(******************************************************************************************************************************************)
(****************************				           Reset Function Part                                                 *****************************)
(******************************************************************************************************************************************)
IF xReset THEN
	xReset:=FALSE;
	xSetEnd:=TRUE;
END_IF;
(******************************************************************************************************************************************)
(****************************				              Error Controlling Part                                            *****************************)
(******************************************************************************************************************************************)
IF (xSetError OR T_Station.TControl.xError) AND NOT(xSetEnd) THEN
	IF NOT(xInitError) THEN
		iStepError:=100;
		xInitError:=TRUE;
		IF NOT(xSetError) THEN
			xSetError:=TRUE;
			xSetTmpError:=FALSE;
		ELSE
			xSetTmpError:=TRUE;
		END_IF;
	END_IF;
	CASE iStepError OF
		100:	IF T_Station.TControl.xError THEN
				diErrorNr:=T_Station.TControl.diErrorNr;
			END_IF;
			IF xSetTmpError THEN
				diErrorNr:=diTmpErrNr;
			END_IF;
			iStepError:=200;
		200:	IF xSetTmpError THEN
				xSetTmpError:=FALSE;
				xStopFctStation1:=FALSE;
				iStepError:=300;
			ELSE
				IF NOT(T_Station.TControl.xError) AND NOT(T_Station.TControl.xEnd) THEN
					IF (T_Station.TControl.iFunctNr = 1) THEN
						T_Station.TControl.xStop:=TRUE;
						xStopFctStation1:=TRUE;
					ELSE
						xStopFctStation1:=FALSE;
					END_IF;
				END_IF;
				iStepError:=300;
			END_IF;
		300:	IF xStopFctStation1 THEN
				IF NOT(T_Station.TControl.xStop) THEN
					xStopFctStation1:=FALSE;
				END_IF;
			END_IF;
			IF NOT(xStopFctStation1) THEN
				xError:=TRUE;
				iStepError:=400;
			END_IF;
		400:	IF xQuitErr THEN
				T_Station.TControl.xQuitError:=T_Station.TControl.xError;
				iStepError:=500;
			END_IF;
		500: IF NOT(T_Station.TControl.xQuitError) THEN
				xSetEnd:=TRUE;
			END_IF;
	END_CASE;
END_IF;
(******************************************************************************************************************************************)
(****************************				              Main Controlling Part                                            *****************************)
(******************************************************************************************************************************************)
IF (xStart OR xStartMainCtr) AND NOT(xSetEnd) AND NOT(xSetError) THEN
	IF NOT (xInitMainCtr) THEN
		iStepPrc:=10;
		xInitMainCtr:=TRUE;
		xStartMainCtr:=TRUE;
		xStart:=FALSE;
		xEnd:=FALSE;
		xSetEndPrc:=FALSE;
		iTmpFunctionNr:=1;
		xAbord:=FALSE;
		T_ExchgParam.T_InfoValueCommon.rActualWireFeedPosition:=0.0;
		T_ExchgParam.T_InfoValueCommon.rActualWireFeedSpeed:=0.0;
	END_IF;
	IF xStop AND NOT(xTmpStop) THEN
		xTmpStop:=TRUE;
		iStepStop:=1;
	END_IF;
	IF xTmpStop THEN
		CASE iStepStop OF
		1:	IF NOT(T_Station.TControl.xEnd) THEN
				T_Station.TControl.xStop:=TRUE;
				iStepStop:=10;
			ELSE
				iStepStop:=20;
			END_IF;
		10:	IF NOT(T_Station.TControl.xStop) THEN
				iStepStop:=20;
			END_IF;
		20:	IF NOT(T_Station.TControl.xStart) AND T_Station.TControl.xEnd THEN
				T_Station.TControl.iFunctNr:=4;
				T_Station.TControl.xStart:=TRUE;
				T_Station.THardware.TAxisGrindFeeder.T_CtrleSingle.lrAcceleration:=T_NovRAMData.T_Standard.T_TeachINGrindFeeder.rAcceleration;
				T_Station.THardware.TAxisGrindFeeder.T_CtrleSingle.lrDecceleration:=T_NovRAMData.T_Standard.T_TeachINGrindFeeder.rDeceleration;
				T_Station.THardware.TAxisGrindFeeder.T_CtrleSingle.lrPosition:=	T_NovRAMData.T_ProcessImageData.T_ProcessPara.rToolDiameterProcess +
																			T_NovRAMData.T_ProcessImageData.T_ProcessPara.rSecurityPosGrindFeedProcess;
				T_Station.THardware.TAxisGrindFeeder.T_CtrleSingle.lrVelocity:=T_NovRAMData.T_ProcessImageData.T_ProcessPara.rSpeedBackwardGrindFeed;
				iStepStop:=30;
			END_IF;
		(* Check Active Movement of the Axis *)
		30:	IF NOT(T_Station.TControl.xStart) AND T_Station.TControl.xEnd THEN
				T_Station.TControl.iFunctNr:=18;	(* Check Axis Movement, and stop it if moves *)
				T_Station.TControl.xStart:=TRUE;
				iStepStop:=40;
			END_IF;
		40:	IF NOT(T_Station.TControl.xStart) AND T_Station.TControl.xEnd THEN
				xStartMainPrc:=FALSE;
				xInitStep:=FALSE;
				iStepPrc:=0;
				xSetEnd:=TRUE;
				RETURN;
			END_IF;
		END_CASE;
		RETURN;
	END_IF;
	IF NOT(xStartMainPrc) THEN
		xStartMainPrc:=TRUE;
	END_IF;
END_IF;
(******************************************************************************************************************************************)
(****************************				             Main Procedure Part                                             *****************************)
(******************************************************************************************************************************************)
IF xStartProcess THEN
	TONStartTimer(IN:=TRUE,PT:=T#1s);
	IF TONStartTimer.Q THEN
		TONStartTimer(IN:=FALSE);
		IF (T_ExchgParam.T_InfoValueCommon.tAutoTimeLeft >= T#1s) THEN
			T_ExchgParam.T_InfoValueCommon.tAutoTimeLeft:=T_ExchgParam.T_InfoValueCommon.tAutoTimeLeft - T#1s;
		ELSE
			T_ExchgParam.T_InfoValueCommon.tAutoTimeLeft:=T#0s;
		END_IF;
	END_IF;
	tStepTime:=T_ExchgParam.T_InfoValueCommon.tAutoTimeTotal / 100;
	TONStartTimer1(IN:=TRUE,PT:=tStepTime);
	IF TONStartTimer1.Q THEN
		TONStartTimer1(IN:=FALSE);
		T_ExchgParam.T_InfoValueCommon.bProgressbarToolCalibration:=T_ExchgParam.T_InfoValueCommon.bProgressbarToolCalibration + 1;
		IF (T_ExchgParam.T_InfoValueCommon.bProgressbarToolCalibration >= 100) THEN
			T_ExchgParam.T_InfoValueCommon.bProgressbarToolCalibration:=100;
		END_IF;
	END_IF;
ELSE
	TONStartTimer(IN:=FALSE);
	TONStartTimer1(IN:=FALSE);
END_IF;
IF xStartMainPrc AND NOT(xSetEnd) AND NOT(xSetError) THEN
	CASE iStepPrc OF
		(* Check first if the ToolCalibration is available to start it *)
		10:	T_Station.THardware.TAxisToolLeft.T_CtrleSingle.lrAcceleration:=T_NovRAMData.T_Standard.T_TeachINToolLeft.rAcceleration;
			T_Station.THardware.TAxisToolLeft.T_CtrleSingle.lrDecceleration:=T_NovRAMData.T_Standard.T_TeachINToolLeft.rDeceleration;
			T_Station.THardware.TAxisToolCenter.T_CtrleSingle.lrAcceleration:=T_NovRAMData.T_Standard.T_TeachINToolCenter.rAcceleration;
			T_Station.THardware.TAxisToolCenter.T_CtrleSingle.lrDecceleration:=T_NovRAMData.T_Standard.T_TeachINToolCenter.rDeceleration;
			T_Station.THardware.TAxisToolRight.T_CtrleSingle.lrAcceleration:=T_NovRAMData.T_Standard.T_TeachINToolRight.rAcceleration;
			T_Station.THardware.TAxisToolRight.T_CtrleSingle.lrDecceleration:=T_NovRAMData.T_Standard.T_TeachINToolRight.rDeceleration;
			T_Station.THardware.TAxisToolFeeder.T_CtrleSingle.lrAcceleration:=T_NovRAMData.T_Standard.T_TeachINToolFeeder.rAcceleration;
			T_Station.THardware.TAxisToolFeeder.T_CtrleSingle.lrDecceleration:=T_NovRAMData.T_Standard.T_TeachINToolFeeder.rDeceleration;
			T_Station.THardware.TAxisGrindFeeder.T_CtrleSingle.lrAcceleration:=T_NovRAMData.T_Standard.T_TeachINGrindFeeder.rAcceleration;
			T_Station.THardware.TAxisGrindFeeder.T_CtrleSingle.lrDecceleration:=T_NovRAMData.T_Standard.T_TeachINGrindFeeder.rDeceleration;
			(* Only for MicroRod, check if the tool is clamped *)
			IF xMicroRodActive THEN
				(*22.12.2009: KFS	{ *)
				(*
				IF T_Station.THardware.TCylToolTension.T_CtrleCyl.xStatePosOn THEN
					xSetError:=TRUE;
					diTmpErrNr:=2;			(* Tool is not clamped *)
				END_IF;
				*)
				(*Added control if all cylinder for the tool are activated*)
				IF T_Station.THardware.TCylToolTension.T_CtrleCyl.xStatePosOn OR
				     T_Station.THardware.TCylToolLeftActive.T_CtrleCyl.T_Standard.xActivOn OR
 				     T_Station.THardware.TCylToolRightActive.T_CtrleCyl.T_Standard.xActivOn  OR
				   (* T_Station.THardware.TCylToolCenterActive.T_CtrleCyl.T_Standard.xActivOn OR*)	(* IGS auskommentiert, diesen Zyl gibts auf der M3 nicht *)
				     NOT(T_Station.THardware.TCylToolPrismaLeftActive.T_CtrleCyl.T_Standard.xActivOn) OR
				     NOT(T_Station.THardware.TCylToolPrismaRightActive.T_CtrleCyl.T_Standard.xActivOn) 	THEN
					xSetError:=TRUE;
					diTmpErrNr:=2;			(* Tool is not clamped *)
				END_IF;
				(*22.12.2009: KFS	} *)
			END_IF;
			(* Only for MicroRod, check if the Machine is referenced *)
			IF xMicroRodActive THEN
				IF NOT(T_Station.TControl.xReferenced) THEN
					xSetError:=TRUE;
					diTmpErrNr:=1;	(* Machine is not referenced *)
					RETURN;
				END_IF;
			END_IF;
			xStartMainPrc:=FALSE;
			xInitStep:=FALSE;
			iStepPrc:=11;
		(* Set the ToolTension force *)
		11:	IF NOT(xInitStep) THEN
				xInitStep:=TRUE;
				T_Station.THardware.TCylToolTension.T_CtrleCyl.iFunction:=2;	(* activate the ToolTension *)
				T_Station.THardware.TCylToolTension.T_CtrleCyl.T_AnalogCylinder.rForceIn:=T_NovRAMData.T_ProcessImageData.T_ProcessPara.rToolTensionProcess;
				IF xMicroRodActive THEN
					T_Station.THardware.TCylToolTension.T_Config.tDelayOn:=T#1s;
				ELSE
					T_Station.THardware.TCylToolTension.T_Config.tDelayOn:=T#0s;
				END_IF;
				T_Station.THardware.TCylToolTension.T_CtrleCyl.xExecute:=TRUE;
			END_IF;
			IF NOT(T_Station.THardware.TCylToolTension.T_CtrleCyl.xExecute) AND T_Station.THardware.TCylToolTension.T_CtrleCyl.xDone THEN
				(* Only for MicroRod, check if the tool is clamped *)
				IF xMicroRodActive THEN
					IF T_Station.THardware.TCylToolTension.T_CtrleCyl.xStatePosOn THEN
						xSetError:=TRUE;
						diTmpErrNr:=2;			(* Tool is not clamped *)
						RETURN;
					END_IF;
				END_IF;
				iStepPrc:=20;
				xStartMainPrc:=FALSE;
				xInitStep:=FALSE;
			END_IF;
		(* Switch First all Axis the power supply on *)
		20:	IF NOT(xInitStep) THEN
				xInitStep:=TRUE;
				T_Station.TControl.iFunctNr:=16;
				T_Station.TControl.xStart:=TRUE;
			END_IF;
			IF NOT(T_Station.TControl.xStart) AND T_Station.TControl.xEnd THEN
				iStepPrc:=30;
				xStartMainPrc:=FALSE;
				xInitStep:=FALSE;
				iTmpStationFunctionNr:=6;
				T_Station.THardware.TAxisToolLeft.T_CtrleSingle.rSetPosition:=0.0;
				T_Station.THardware.TAxisToolCenter.T_CtrleSingle.rSetPosition:=0.0;
				T_Station.THardware.TAxisToolRight.T_CtrleSingle.rSetPosition:=0.0;
				T_Station.THardware.TAxisToolFeeder.T_CtrleSingle.rSetPosition:=0.0;
			END_IF;
		(* Reset the Position of the Axis *)
		30:	IF NOT(xInitStep) THEN
				xInitStep:=TRUE;
				(* 6=ToolLeft, 7=ToolCenter, 8=ToolRight, 9=ToolFeeder *)
				T_Station.TControl.iFunctNr:=iTmpStationFunctionNr;
				T_Station.TControl.xStart:=TRUE;
			END_IF;
			IF NOT(T_Station.TControl.xStart) AND T_Station.TControl.xEnd THEN
				iTmpStationFunctionNr:=iTmpStationFunctionNr + 1;
				IF NOT(xMicroRodActive) AND (iTmpStationFunctionNr = 7) THEN
					iTmpStationFunctionNr:=iTmpStationFunctionNr + 1;
				END_IF;
				IF xMicroRodActive AND (iTmpStationFunctionNr = 9) THEN
					iTmpStationFunctionNr:=iTmpStationFunctionNr + 1;
				END_IF;
				xStartMainPrc:=FALSE;
				xInitStep:=FALSE;
				IF (iTmpStationFunctionNr < 10) THEN
					iStepPrc:=30;
				ELSE
					iStepPrc:=40;
				END_IF;
			END_IF;
		(* GrindFeeder Set Absolut to Security Position *)
		40:	IF NOT(xInitStep) THEN
				xInitStep:=TRUE;
				T_Station.TControl.iFunctNr:=4;
				T_Station.TControl.xStart:=TRUE;
				T_Station.THardware.TAxisGrindFeeder.T_CtrleSingle.lrAcceleration:=T_NovRAMData.T_Standard.T_TeachINGrindFeeder.rAcceleration;
				T_Station.THardware.TAxisGrindFeeder.T_CtrleSingle.lrDecceleration:=T_NovRAMData.T_Standard.T_TeachINGrindFeeder.rDeceleration;
				T_Station.THardware.TAxisGrindFeeder.T_CtrleSingle.lrPosition:=	T_NovRAMData.T_ProcessImageData.T_ProcessPara.rToolDiameterProcess +
																			T_NovRAMData.T_ProcessImageData.T_ProcessPara.rSecurityPosGrindFeedProcess;
				T_Station.THardware.TAxisGrindFeeder.T_CtrleSingle.lrVelocity:=T_NovRAMData.T_ProcessImageData.T_ProcessPara.rSpeedBackwardGrindFeed;
			END_IF;
			IF NOT(T_Station.TControl.xStart) AND T_Station.TControl.xEnd THEN
				IF xMicroRodActive THEN
					iStepPrc:=50;
				ELSE
					iStepPrc:=60;
				END_IF;
				xStartMainPrc:=FALSE;
				xInitStep:=FALSE;
			END_IF;
		(* Only for MicroRod-->Set ToolFeed Absolut to the StartPosition and if more cycle than only the first time *)
		50:	IF NOT(xInitStep) THEN
				xInitStep:=TRUE;
				T_Station.TControl.iFunctNr:=14;
				T_Station.TControl.xStart:=TRUE;
				T_Station.THardware.TAxisToolFeeder.T_CtrleSingle.lrAcceleration:=T_NovRAMData.T_Standard.T_TeachINToolFeeder.rAcceleration;
				T_Station.THardware.TAxisToolFeeder.T_CtrleSingle.lrDecceleration:=T_NovRAMData.T_Standard.T_TeachINToolFeeder.rDeceleration;
				T_Station.THardware.TAxisToolFeeder.T_CtrleSingle.lrPosition:=T_NovRAMData.T_ProcessImageData.T_CalibrationPara.rStartPosToolFeedCalib;
				T_Station.THardware.TAxisToolFeeder.T_CtrleSingle.lrVelocity:=T_NovRAMData.T_ProcessImageData.T_ProcessPara.rSpeedStartPosToolFeedProcess;
			END_IF;
			IF NOT(T_Station.TControl.xStart) AND T_Station.TControl.xEnd THEN
				iStepPrc:=60;
				xStartMainPrc:=FALSE;
				xInitStep:=FALSE;
			END_IF;
		(* ToolRotation Start *)
		60:	IF NOT(xInitStep) THEN
				xInitStep:=TRUE;
				T_Station.TControl.iFunctNr:=2;
				T_Station.TControl.xStart:=TRUE;
				(* ToolLeft --> Master *)
				T_Station.THardware.TAxisToolLeft.T_CtrleSingle.lrVelocity:=T_NovRAMData.T_ProcessImageData.T_CalibrationPara.rSpeedToolRotationCalib;
				T_Station.THardware.TAxisToolLeft.T_CtrleSingle.lrAcceleration:=T_NovRAMData.T_Standard.T_TeachINToolLeft.rAcceleration;
				T_Station.THardware.TAxisToolLeft.T_CtrleSingle.lrDecceleration:=T_NovRAMData.T_Standard.T_TeachINToolLeft.rDeceleration;
				IF xMicroRodActive THEN
					(* ToolCenter --> Slave of ToolLeft only by MicroRod *)
					T_Station.THardware.TAxisToolCenter.T_CtrleSingle.lrAcceleration:=T_NovRAMData.T_Standard.T_TeachINToolCenter.rAcceleration;
					T_Station.THardware.TAxisToolCenter.T_CtrleSingle.lrDecceleration:=T_NovRAMData.T_Standard.T_TeachINToolCenter.rDeceleration;
					T_Station.THardware.TAxisToolCenter.T_CtrleSingle.lrGearDivider:=INT_TO_LREAL(T_Station.T_WorkTool.iBaseGearDivider);
					T_Station.THardware.TAxisToolCenter.T_CtrleSingle.lrGearFactor:=(	INT_TO_LREAL(T_Station.T_WorkTool.iBaseGearDivider) /
																					(T_Station.THardware.TAxisToolLeft.T_CtrleSingle.lrGearRatio /
																					T_Station.THardware.TAxisToolCenter.T_CtrleSingle.lrGearRatio)) * -1.0;

					(* ToolRight --> Slave of ToolLeft by MicroWire or Slave of ToolRight by MicroRod *)
					T_Station.THardware.TAxisToolRight.T_CtrleSingle.lrAcceleration:=T_NovRAMData.T_Standard.T_TeachINToolRight.rAcceleration;
					T_Station.THardware.TAxisToolRight.T_CtrleSingle.lrDecceleration:=T_NovRAMData.T_Standard.T_TeachINToolRight.rDeceleration;
					T_Station.THardware.TAxisToolRight.T_CtrleSingle.lrGearDivider:=INT_TO_LREAL(T_Station.T_WorkTool.iBaseGearDivider);
					T_Station.THardware.TAxisToolRight.T_CtrleSingle.lrGearFactor:=	INT_TO_LREAL(T_Station.T_WorkTool.iBaseGearDivider) /
																					(T_Station.THardware.TAxisToolLeft.T_CtrleSingle.lrGearRatio /
																					T_Station.THardware.TAxisToolRight.T_CtrleSingle.lrGearRatio);
				END_IF;

				IF NOT(xMicroRodActive) THEN
					(* ToolRight --> Slave of ToolRight by MicroWire *)
					T_Station.THardware.TAxisToolFeeder.T_CtrleSingle.lrAcceleration:=T_NovRAMData.T_Standard.T_TeachINToolFeeder.rAcceleration;
					T_Station.THardware.TAxisToolFeeder.T_CtrleSingle.lrDecceleration:=T_NovRAMData.T_Standard.T_TeachINToolFeeder.rDeceleration;
					T_Station.THardware.TAxisToolFeeder.T_CtrleSingle.lrGearDivider:=INT_TO_LREAL(T_Station.T_WorkTool.iBaseGearDivider);
					T_Station.THardware.TAxisToolFeeder.T_CtrleSingle.lrGearFactor:=	(INT_TO_LREAL(T_Station.T_WorkTool.iBaseGearDivider) /
																					(T_Station.THardware.TAxisToolFeeder.T_CtrleSingle.lrGearRatio /
																					T_Station.THardware.TAxisToolRight.T_CtrleSingle.lrGearRatio)) * -1.0;

					(* ToolRight --> Slave of ToolLeft by MicroWire or Slave of ToolRight by MicroRod *)
					T_Station.THardware.TAxisToolRight.T_CtrleSingle.lrAcceleration:=T_NovRAMData.T_Standard.T_TeachINToolRight.rAcceleration;
					T_Station.THardware.TAxisToolRight.T_CtrleSingle.lrDecceleration:=T_NovRAMData.T_Standard.T_TeachINToolRight.rDeceleration;
					T_Station.THardware.TAxisToolRight.T_CtrleSingle.lrGearDivider:=INT_TO_LREAL(T_Station.T_WorkTool.iBaseGearDivider);
					T_Station.THardware.TAxisToolRight.T_CtrleSingle.lrGearFactor:=	(INT_TO_LREAL(T_Station.T_WorkTool.iBaseGearDivider) /
																					(T_Station.THardware.TAxisToolLeft.T_CtrleSingle.lrGearRatio /
																					T_Station.THardware.TAxisToolRight.T_CtrleSingle.lrGearRatio)) * -1.0;
				END_IF;
			END_IF;
			IF NOT(T_Station.TControl.xStart) AND T_Station.TControl.xEnd THEN
				xStartMainPrc:=FALSE;
				xInitStep:=FALSE;
				iStepPrc:=70;
			END_IF;
		(* GrindFeeder Set Absolut to ToolDiameter minus the offset with the fast speed *)
		70:	IF NOT(xInitStep) THEN
				xInitStep:=TRUE;
				T_Station.TControl.iFunctNr:=4;
				T_Station.TControl.xStart:=TRUE;
				T_Station.THardware.TAxisGrindFeeder.T_CtrleSingle.lrAcceleration:=T_NovRAMData.T_Standard.T_TeachINGrindFeeder.rAcceleration;
				T_Station.THardware.TAxisGrindFeeder.T_CtrleSingle.lrDecceleration:=T_NovRAMData.T_Standard.T_TeachINGrindFeeder.rDeceleration;
				T_Station.THardware.TAxisGrindFeeder.T_CtrleSingle.lrPosition:=T_NovRAMData.T_ProcessImageData.T_ProcessPara.rToolDiameterProcess + T_NovRAMData.T_ProcessImageData.T_ProcessPara.rOffsetBeforeToolDiaGrindFeedProcess;
				T_Station.THardware.TAxisGrindFeeder.T_CtrleSingle.lrVelocity:=T_NovRAMData.T_ProcessImageData.T_ProcessPara.rSpeedForwardFastGrindFeed;
			END_IF;
			IF NOT(T_Station.TControl.xStart) AND T_Station.TControl.xEnd THEN
				xStartMainPrc:=FALSE;
				xInitStep:=FALSE;
				iStepPrc:=80;
			END_IF;
		(* Working ToolCalibration *)
		80:	IF NOT(xInitStep) THEN
				xStartProcess:=TRUE;
				xInitStep:=TRUE;
				T_Station.TControl.iFunctNr:=13;
				T_Station.TControl.xStart:=TRUE;
			END_IF;
			IF NOT(T_Station.TControl.xStart) AND T_Station.TControl.xEnd THEN
				xStartMainPrc:=FALSE;
				xInitStep:=FALSE;
				iStepPrc:=90;
				RETURN;
			END_IF;
			(* Only for MicroRod, check if the tool is clamped *)
			IF xMicroRodActive THEN
				IF T_Station.THardware.TCylToolTension.T_CtrleCyl.xStatePosOn THEN
					xStartMainPrc:=FALSE;
					xInitStep:=FALSE;
					iStepPrc:=81;
					RETURN;
				END_IF;
			END_IF;
		(* Stop the Process, because the Tool is broken *)
		81:	IF NOT(xInitStep) THEN
				xInitStep:=TRUE;
				T_Station.TControl.xStop:=TRUE;
			END_IF;
			IF NOT(T_Station.TControl.xStart) AND T_Station.TControl.xEnd THEN
				xStartMainPrc:=FALSE;
				xInitStep:=FALSE;
				iStepPrc:=82;
			END_IF;
		(* Set the GrindFeeder to the security Position *)
		82:	IF NOT(xInitStep) THEN
				xInitStep:=TRUE;
				T_Station.TControl.iFunctNr:=4;
				T_Station.TControl.xStart:=TRUE;
				T_Station.THardware.TAxisGrindFeeder.T_CtrleSingle.lrAcceleration:=T_NovRAMData.T_Standard.T_TeachINGrindFeeder.rAcceleration;
				T_Station.THardware.TAxisGrindFeeder.T_CtrleSingle.lrDecceleration:=T_NovRAMData.T_Standard.T_TeachINGrindFeeder.rDeceleration;
				T_Station.THardware.TAxisGrindFeeder.T_CtrleSingle.lrPosition:=	T_NovRAMData.T_ProcessImageData.T_ProcessPara.rToolDiameterProcess +
																			T_NovRAMData.T_ProcessImageData.T_ProcessPara.rSecurityPosGrindFeedProcess;
				T_Station.THardware.TAxisGrindFeeder.T_CtrleSingle.lrVelocity:=T_NovRAMData.T_ProcessImageData.T_ProcessPara.rSpeedBackwardGrindFeed;
			END_IF;
			IF NOT(T_Station.TControl.xStart) AND T_Station.TControl.xEnd THEN
				xStartMainPrc:=FALSE;
				xInitStep:=FALSE;
				iStepPrc:=83;
			END_IF;
		(* Check Active Movement of the Axis *)
		83:	IF NOT(xInitStep) THEN
				xInitStep:=TRUE;
				T_Station.TControl.iFunctNr:=18;	(* Check Axis Movement, and stop it if moves *)
				T_Station.TControl.xStart:=TRUE;
			END_IF;
			IF NOT(T_Station.TControl.xStart) AND T_Station.TControl.xEnd THEN
				xSetError:=TRUE;
				diTmpErrNr:=2;			(* Tool is not clamped *)
				RETURN;
			END_IF;
		(* GrindFeeder Set Absolut to Security Position *)
		90:	IF NOT(xInitStep) THEN
				xInitStep:=TRUE;
				T_Station.TControl.iFunctNr:=4;
				T_Station.TControl.xStart:=TRUE;
				T_Station.THardware.TAxisGrindFeeder.T_CtrleSingle.lrAcceleration:=T_NovRAMData.T_Standard.T_TeachINGrindFeeder.rAcceleration;
				T_Station.THardware.TAxisGrindFeeder.T_CtrleSingle.lrDecceleration:=T_NovRAMData.T_Standard.T_TeachINGrindFeeder.rDeceleration;
				T_Station.THardware.TAxisGrindFeeder.T_CtrleSingle.lrPosition:=	T_NovRAMData.T_ProcessImageData.T_ProcessPara.rToolDiameterProcess +
																			T_NovRAMData.T_ProcessImageData.T_ProcessPara.rSecurityPosGrindFeedProcess;
				T_Station.THardware.TAxisGrindFeeder.T_CtrleSingle.lrVelocity:=T_NovRAMData.T_ProcessImageData.T_ProcessPara.rSpeedBackwardGrindFeed;
			END_IF;
			IF NOT(T_Station.TControl.xStart) AND T_Station.TControl.xEnd THEN
				xStartMainPrc:=FALSE;
				xInitStep:=FALSE;
				iStepPrc:=100;
			END_IF;
		(* ToolRotation Stop *)
		100:	IF NOT(xInitStep) THEN
				xInitStep:=TRUE;
				T_Station.TControl.iFunctNr:=3;
				T_Station.TControl.xStart:=TRUE;
				(* ToolLeft --> Master *)
				T_Station.THardware.TAxisToolLeft.T_CtrleSingle.lrAcceleration:=T_NovRAMData.T_Standard.T_TeachINToolLeft.rAcceleration;
				T_Station.THardware.TAxisToolLeft.T_CtrleSingle.lrDecceleration:=T_NovRAMData.T_Standard.T_TeachINToolLeft.rDeceleration;
				IF xMicroRodActive THEN
					(* ToolCenter --> Slave of ToolLeft only by MicroRod *)
					T_Station.THardware.TAxisToolCenter.T_CtrleSingle.lrAcceleration:=T_NovRAMData.T_Standard.T_TeachINToolCenter.rAcceleration;
					T_Station.THardware.TAxisToolCenter.T_CtrleSingle.lrDecceleration:=T_NovRAMData.T_Standard.T_TeachINToolCenter.rDeceleration;
				END_IF;
				(* ToolRight --> Slave of ToolLeft by MicroWire or Slave of ToolRight by MicroRod *)
				T_Station.THardware.TAxisToolRight.T_CtrleSingle.lrAcceleration:=T_NovRAMData.T_Standard.T_TeachINToolRight.rAcceleration;
				T_Station.THardware.TAxisToolRight.T_CtrleSingle.lrDecceleration:=T_NovRAMData.T_Standard.T_TeachINToolRight.rDeceleration;
				IF NOT(xMicroRodActive) THEN
					(* ToolRight --> Slave of ToolRight by MicroWire *)
					T_Station.THardware.TAxisToolFeeder.T_CtrleSingle.lrAcceleration:=T_NovRAMData.T_Standard.T_TeachINToolFeeder.rAcceleration;
					T_Station.THardware.TAxisToolFeeder.T_CtrleSingle.lrDecceleration:=T_NovRAMData.T_Standard.T_TeachINToolFeeder.rDeceleration;
				END_IF;
			END_IF;
			IF NOT(T_Station.TControl.xStart) AND T_Station.TControl.xEnd THEN
				xStartMainPrc:=FALSE;
				xInitStep:=FALSE;
				iStepPrc:=110;
			END_IF;
		110:	xSetEndPrc:=FALSE;
			xStartMainPrc:=FALSE;
			xInitStep:=FALSE;
			iStepPrc:=0;
			xSetEnd:=TRUE;
	END_CASE;
END_IF;
(******************************************************************************************************************************************)
(****************************				             	Init / Reset Part                                                   *****************************)
(******************************************************************************************************************************************)
IF xSetEnd THEN
	xEnd:=TRUE;
	xInitStep:=FALSE;
	xSetEnd:=FALSE;
	xStop:=FALSE;
	xStartMainPrc:=FALSE;
	xTmpStop:=FALSE;
	xInitMainCtr:=FALSE;
	xStartMainCtr:=FALSE;
	xStart:=FALSE;
	xSetError:=FALSE;
	xQuitErr:=FALSE;
	xError:=FALSE;
	diErrorNr:=0;
	xInitError:=FALSE;
	xFreeze:=FALSE;
	xAbord:=FALSE;
	xTmpAbord:=FALSE;
	xSetEndPrc:=FALSE;
	xStartProcess:=FALSE;
END_IF;
END_FUNCTION_BLOCK

(* POU PRG_STATION_LAYER3/PRG_STATION, FBD *)
PROGRAM PRG_STATION
VAR
	FBStation: FB_STATION;
END_VAR
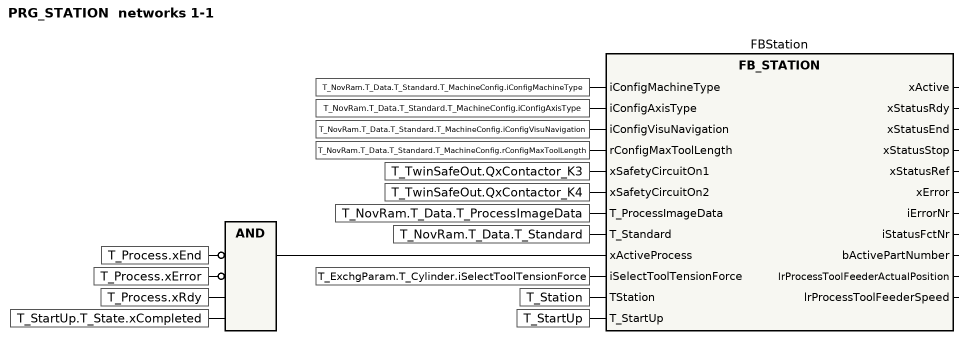
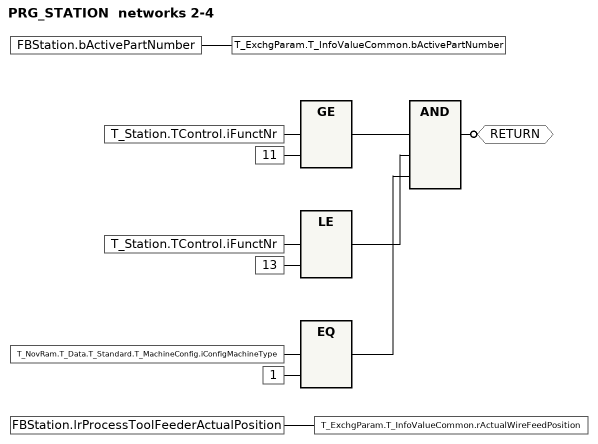
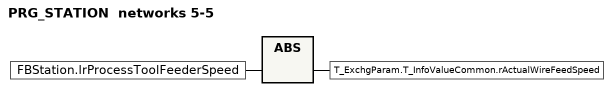
_FBD_ (* Function Block Diagram *)
NETWORK 1 (* STATION LEVEL-->LAYER 3 *)
	FBStation:FB_STATION(iConfigMachineType: T_NovRam.T_Data.T_Standard.T_MachineConfig.iConfigMachineType, iConfigAxisType: T_NovRam.T_Data.T_Standard.T_MachineConfig.iConfigAxisType, iConfigVisuNavigation: T_NovRam.T_Data.T_Standard.T_MachineConfig.iConfigVisuNavigation, rConfigMaxToolLength: T_NovRam.T_Data.T_Standard.T_MachineConfig.rConfigMaxToolLength, xSafetyCircuitOn1: T_TwinSafeOut.QxContactor_K3, xSafetyCircuitOn2: T_TwinSafeOut.QxContactor_K4, T_ProcessImageData: T_NovRam.T_Data.T_ProcessImageData, T_Standard: T_NovRam.T_Data.T_Standard, xActiveProcess: AND(NOT T_Process.xEnd, NOT T_Process.xError, T_Process.xRdy, T_StartUp.T_State.xCompleted), iSelectToolTensionForce: T_ExchgParam.T_Cylinder.iSelectToolTensionForce, TStation: T_Station, T_StartUp: T_StartUp)
NETWORK 2
	FBStation.bActivePartNumber => T_ExchgParam.T_InfoValueCommon.bActivePartNumber
NETWORK 3
	NOT AND(GE(T_Station.TControl.iFunctNr, 11), LE(T_Station.TControl.iFunctNr, 13), EQ(T_NovRam.T_Data.T_Standard.T_MachineConfig.iConfigMachineType, 1)) => <RETURN>
NETWORK 4
	FBStation.lrProcessToolFeederActualPosition => T_ExchgParam.T_InfoValueCommon.rActualWireFeedPosition
NETWORK 5
	ABS(FBStation.lrProcessToolFeederSpeed) => T_ExchgParam.T_InfoValueCommon.rActualWireFeedSpeed
_END_FBD_
(* the same logic as Structured Text *)
(* Network 1: STATION LEVEL-->LAYER 3 *)
FBStation(iConfigMachineType := T_NovRam.T_Data.T_Standard.T_MachineConfig.iConfigMachineType, iConfigAxisType := T_NovRam.T_Data.T_Standard.T_MachineConfig.iConfigAxisType, iConfigVisuNavigation := T_NovRam.T_Data.T_Standard.T_MachineConfig.iConfigVisuNavigation, rConfigMaxToolLength := T_NovRam.T_Data.T_Standard.T_MachineConfig.rConfigMaxToolLength, xSafetyCircuitOn1 := T_TwinSafeOut.QxContactor_K3, xSafetyCircuitOn2 := T_TwinSafeOut.QxContactor_K4, T_ProcessImageData := T_NovRam.T_Data.T_ProcessImageData, T_Standard := T_NovRam.T_Data.T_Standard, xActiveProcess := NOT T_Process.xEnd AND NOT T_Process.xError AND T_Process.xRdy AND T_StartUp.T_State.xCompleted, iSelectToolTensionForce := T_ExchgParam.T_Cylinder.iSelectToolTensionForce, TStation := T_Station, T_StartUp := T_StartUp);
(* Network 2 *)
T_ExchgParam.T_InfoValueCommon.bActivePartNumber := FBStation.bActivePartNumber;
(* Network 3 *)
IF NOT ((T_Station.TControl.iFunctNr >= 11) AND (T_Station.TControl.iFunctNr <= 13) AND (T_NovRam.T_Data.T_Standard.T_MachineConfig.iConfigMachineType = 1)) THEN RETURN; END_IF;
(* Network 4 *)
T_ExchgParam.T_InfoValueCommon.rActualWireFeedPosition := FBStation.lrProcessToolFeederActualPosition;
(* Network 5 *)
T_ExchgParam.T_InfoValueCommon.rActualWireFeedSpeed := ABS(FBStation.lrProcessToolFeederSpeed);
END_PROGRAM

(* POU PRG_STATION_LAYER3/FB_STATIONEN/FB_FUNCTION/FB_STATION, ST *)
FUNCTION_BLOCK FB_STATION
VAR_INPUT
	iConfigMachineType:INT;
	iConfigAxisType:INT;
	iConfigVisuNavigation:INT;
	rConfigMaxToolLength:REAL;
	xSafetyCircuitOn1:BOOL;
	xSafetyCircuitOn2:BOOL;
	T_ProcessImageData:ST_RETAIN_DATA_PROCESSIMAGE;
	T_Standard:ST_RETAIN_DATA;
	xActiveProcess:BOOL;
	iSelectToolTensionForce:INT;
END_VAR
VAR_IN_OUT
	TStation:ST_STATION;
	T_StartUp:ST_STARTUP;
END_VAR
VAR_OUTPUT
	xActive : BOOL :=FALSE;
	xStatusRdy : BOOL := FALSE;
	xStatusEnd : BOOL := FALSE;
	xStatusStop : BOOL := FALSE;
	xStatusRef : BOOL := FALSE;
	xError : BOOL := FALSE;
	iErrorNr : DINT :=0;
	iStatusFctNr : INT := 0;
	bActivePartNumber:BYTE;
	lrProcessToolFeederActualPosition:LREAL;
	lrProcessToolFeederSpeed:LREAL;
END_VAR
VAR
(* Pointer auf Actuatoren *)
	ptrTAxisToolLeft:POINTER TO ST_AXIS;
	ptrTAxisToolCenter:POINTER TO ST_AXIS;
	ptrTAxisToolRight:POINTER TO ST_AXIS;
	ptrTAxisToolFeeder:POINTER TO ST_AXIS;
	ptrTAxisGrindFeeder:POINTER TO ST_AXIS;
	ptrTAxisGrindSpindle:POINTER TO ST_AXIS;			(* IGS *)
	ptrTCylToolTension:POINTER TO ST_CYLINDER;
(*22.12.2009: KFS {    *)
	ptrTCylToolLeftActive:POINTER TO ST_CYLINDER;
	ptrTCylToolRightActive:POINTER TO ST_CYLINDER;
	ptrTCylToolCenterActive:POINTER TO ST_CYLINDER;
	ptrTCylToolPrismaLeftActive:POINTER TO ST_CYLINDER;
	ptrTCylToolPrismaRightActive:POINTER TO ST_CYLINDER;
	ptrTToolFeederWorkLength:POINTER TO ST_CYLINDER;
(*22.12.2009: KFS }   *)
	ptrTFunction:POINTER TO ST_CTRL_FUNCTION;
	xSetEnableConfig: BOOL;
	iEnableConfigMachineType:INT;
	iTmpConfigMachineType:INT;
	iEnableConfigAxisType:INT;
	iTmpConfigAxisType:INT;
	iEnableConfigVisuNavigation:INT;
	iTmpConfigVisuNavigation:INT;
	rEnableConfigMaxToolLength:REAL;
	rTmpConfigMaxToolLength:REAL;
	xMicroRodActive: BOOL;
	xBeckhoffDriveActive: BOOL;
	xTmpStopFunction: BOOL;
	iStationFunctionNr: INT;
	xStartFunction: BOOL := FALSE;
	xTmpStart: BOOL := FALSE;
	xInitStart: BOOL := FALSE;
	xSetEnd: BOOL := FALSE;
	xInitError: BOOL := FALSE;
	xInitStop: BOOL := FALSE;
	xInitSetEnable: BOOL := FALSE;
	iStepEnable: INT := 0;
	xInitStep: BOOL := FALSE;
	iAxisFunctionNr: INT :=0;
	xInitDelEnable: BOOL := FALSE;
	xStationError: BOOL := FALSE;
	xStepError: BOOL;
	iStepError: INT;
	xTmpStationError: BOOL;
	xRdyDisableStation: BOOL;
	xReadyChkError: BOOL;
	xDontDeleteErrorFlag: BOOL;
	xSetError: BOOL;
(* Trigger *)
	fbFTrig: F_TRIG;
	fbRTrig: R_TRIG;
	xTmp: BOOL;
	diErrorNumber: DINT;
	iCountCycle: INT;
	xSecurityCircuitOn: BOOL;
	xSecurityCircuitOff: BOOL;
	iStepSecCircuit: INT;
	xInitSecCircuit: BOOL;
	TONCheckTimeOut: TON;
	xPowerSwitchedOn: BOOL;
	xChkConfigStation: BOOL;
	FBFctToolRotationTorqueStart: FB_FctToolRotationTorqueStart;
	FBFctToolRotationTorqueStop: FB_FctToolRotationTorqueStop;
	FBFctGrindFeedAbsRelPosition: FB_FctGrindFeedAbsRelPosition;
	FBFctSetAxisPosition: FB_FctSetAxisPosition;
	FBFctToolWorkingGeometry: FB_FctToolWorkingGeometry;
	FBFctToolWorkingGeometryMultiCycle: FB_FctToolWorkingGeometryMultiCycle;
	FBFctToolWorkingGroove: FB_FctToolWorkingGroove;
	FBFctToolCalibration: FB_FctToolCalibration;
	iMaxFunctionNr:INT:=20;
	(* 17.11.2010 KFS : iMaxFunctionNr:INT:=19*)
	FBFctToolFeedAbsRelPosition: FB_FctToolFeedAbsRelPosition;
	FBFctSwitchOnOffPowerSupply: FB_FctSwitchOnOffPowerSupply;
	(* 17.11.2010: KFS 	{	*)
	FBFctToolFeedMaxLenReference:FB_FctToolFeedMaxLenReference;
	(* 17.11.2010: KFS 	}	*)
	FBFctToolFeedReference: FB_FctToolFeedReference;
	xCheckAxisError: BOOL;
	xFirstTimeBooting: BOOL:=FALSE;
	FBFctStopAxisMovement: FB_FctStopAxisMovement;
	xAxisErrorActive: BOOL;
	xWaitSetError: BOOL;
	TONWaitSetError: TON;
	xForceHWError: BOOL;
	xCheckActiveFunction: BOOL;
	xForceResetAxis: BOOL;
	xReadyToQuitErr: BOOL;
	TONWaitReset: TON;
END_VAR
(****************************************************************************************************************************************************)
(***********                 This Functionblock manage all the station funtion and synchronizing of the Hardware                           ************)
(****************************************************************************************************************************************************)
xActive:=TStation.TControl.xActiveStation;
IF NOT(TStation.TControl.xActiveStation) THEN
	(*TStation:=TDeleteStationStruct;*)
	RETURN;
ELSE
	IF xSetEnableConfig THEN
		IF (iEnableConfigMachineType <> iConfigMachineType) THEN
			iTmpConfigMachineType:=iEnableConfigMachineType;
		ELSE
			iTmpConfigMachineType:=iConfigMachineType;
		END_IF;
		IF (iEnableConfigAxisType <> iConfigAxisType) THEN
			iTmpConfigAxisType:=iEnableConfigAxisType;
		ELSE
			iTmpConfigAxisType:=iConfigAxisType;
		END_IF;
		IF (iEnableConfigVisuNavigation <> iConfigVisuNavigation) THEN
			iTmpConfigVisuNavigation:=iEnableConfigVisuNavigation;
		ELSE
			iTmpConfigVisuNavigation:=iConfigVisuNavigation;
		END_IF;
		IF (rEnableConfigMaxToolLength <> rConfigMaxToolLength) THEN
			rTmpConfigMaxToolLength:=rEnableConfigMaxToolLength;
		ELSE
			rTmpConfigMaxToolLength:=rConfigMaxToolLength;
		END_IF;
		(*08.12.2010 KFS:	{	*)
		IF T_Station.xOverwriteMaxToolLength THEN
			rEnableConfigMaxToolLength:=rConfigMaxToolLength;
			rTmpConfigMaxToolLength:=rConfigMaxToolLength;
		END_IF;
		(*08.12.2010 KFS:	}	*)
	ELSE
		iTmpConfigMachineType:=iConfigMachineType;
		iTmpConfigAxisType:=iConfigAxisType;
		iTmpConfigVisuNavigation:=iConfigVisuNavigation;
		rTmpConfigMaxToolLength:=rConfigMaxToolLength;
	END_IF;
	(* Zuweisung der Datenstrukturen der Aktuatoren als Pointer *)
	ptrTAxisToolLeft:=ADR(TStation.THardware.TAxisToolLeft);
	ptrTAxisToolCenter:=ADR(TStation.THardware.TAxisToolCenter);
	ptrTAxisToolRight:=ADR(TStation.THardware.TAxisToolRight);
	ptrTAxisToolFeeder:=ADR(TStation.THardware.TAxisToolFeeder);
	ptrTAxisGrindFeeder:=ADR(TStation.THardware.TAxisGrindFeeder);
	ptrTAxisGrindSpindle:=ADR(TStation.THardware.TAxisGrindSpindle);
	ptrTCylToolTension:=ADR(TStation.THardware.TCylToolTension);
(*22.12.2009: KFS {    *)
	ptrTCylToolLeftActive:=ADR(TStation.THardware.TCylToolLeftActive);
	ptrTCylToolRightActive:=ADR(TStation.THardware.TCylToolRightActive);
	ptrTCylToolCenterActive:=ADR(TStation.THardware.TCylToolCenterActive);
	ptrTCylToolPrismaLeftActive:=ADR(TStation.THardware.TCylToolPrismaLeftActive);
	ptrTCylToolPrismaRightActive:=ADR(TStation.THardware.TCylToolPrismaRightActive);
	ptrTToolFeederWorkLength:=ADR(TStation.THardware.TToolFeederWorkLength);
(*22.12.2009: KFS }   *)
	ptrTFunction:=ADR(TStation.TCtrlFunction);
	IF (iConfigMachineType = 2) THEN
		xMicroRodActive:=TRUE;
	ELSE
		xMicroRodActive:=FALSE;
	END_IF;
	IF (iConfigAxisType = 2) THEN
		xBeckhoffDriveActive:=TRUE;
	ELSE
		xBeckhoffDriveActive:=FALSE;
	END_IF;
	IF xSafetyCircuitOn1 AND xSafetyCircuitOn2 THEN
		xPowerSwitchedOn:=TRUE;
	ELSE
		xPowerSwitchedOn:=FALSE;
	END_IF;
END_IF;
(******************************************************************************************************************************************)
(****************************				                  Status Part                                                            *****************************)
(******************************************************************************************************************************************)
xStatusRdy:=TStation.TControl.xRdy;
xStatusEnd:=TStation.TControl.xEnd;
xStatusStop:=xTmpStopFunction;
IF xMicroRodActive THEN
	TStation.TControl.xReferenced:=ptrTAxisToolFeeder^.T_CtrleSingle.xRef;
ELSE
	TStation.TControl.xReferenced:=TRUE;
END_IF;
xStatusRef:=TStation.TControl.xReferenced;
xError:= TStation.TControl.xError;
iErrorNr := TStation.TControl.diErrorNr;
iStatusFctNr:=iStationFunctionNr;
(******************************************************************************************************************************************)
(****************************				                Enable & Disable Part                                                            *****************************)
(******************************************************************************************************************************************)
(* Check Active of the Axis Drives *)
xTmp:=	(NOT(ptrTAxisToolLeft^.T_CtrleSingle.xErr) AND NOT(ptrTAxisToolLeft^.T_CtrleSingle.xDone)) OR
		(NOT(ptrTAxisToolCenter^.T_CtrleSingle.xErr) AND NOT(ptrTAxisToolCenter^.T_CtrleSingle.xDone) AND xMicroRodActive) OR
		(NOT(ptrTAxisToolRight^.T_CtrleSingle.xErr) AND NOT(ptrTAxisToolRight^.T_CtrleSingle.xDone)) OR
		(NOT(ptrTAxisToolFeeder^.T_CtrleSingle.xErr) AND NOT(ptrTAxisToolFeeder^.T_CtrleSingle.xDone)) OR
		(NOT(ptrTAxisGrindFeeder^.T_CtrleSingle.xErr) AND NOT(ptrTAxisGrindFeeder^.T_CtrleSingle.xDone)) OR
		(NOT(ptrTAxisGrindSpindle^.T_CtrleSingle.xErr) AND NOT(ptrTAxisGrindSpindle^.T_CtrleSingle.xDone));
CtrlDisableStation;
CtrlEnableStation;



(******************************************************************************************************************************************)
(****************************				       Security Circuit Switch ON/OFF                                          *****************************)
(******************************************************************************************************************************************)
CtrlSafetySwitch_ON_OFF;


(******************************************************************************************************************************************)
(****************************				         Error Controlling Part                                                  *****************************)
(******************************************************************************************************************************************)
IF xActiveProcess THEN
	IF (ptrTAxisToolLeft^.T_CtrleSingle.xErr OR (ptrTAxisToolCenter^.T_CtrleSingle.xErr AND xMicroRodActive) OR ptrTAxisToolRight^.T_CtrleSingle.xErr OR
              ptrTAxisToolFeeder^.T_CtrleSingle.xErr OR ptrTAxisGrindFeeder^.T_CtrleSingle.xErr) AND NOT(xWaitSetError) THEN
		xWaitSetError:=TRUE;
		TONWaitSetError(IN:=FALSE);
	END_IF;
	IF xWaitSetError THEN
		TONWaitSetError(IN:=TRUE,PT:=T#50ms);
		IF TONWaitSetError.Q THEN
			xForceHWError:=TRUE;
		END_IF;
	END_IF;
ELSE
	xWaitSetError:=FALSE;
	xForceHWError:=FALSE;
	TONWaitSetError(IN:=FALSE);
END_IF;
CtrlErrorStation;


(******************************************************************************************************************************************)
(****************************				         Main Controlling Part                                                  *****************************)
(******************************************************************************************************************************************)
CtrlMainStation;


(******************************************************************************************************************************************)
(****************************				   Check Configuration Station Part                                 *****************************)
(******************************************************************************************************************************************)
IF (xStartFunction OR xChkConfigStation) AND xSetEnableConfig THEN
	IF NOT(xChkConfigStation) THEN
		IF (iEnableConfigMachineType <> iConfigMachineType) OR (iEnableConfigAxisType <> iConfigAxisType) OR (iEnableConfigVisuNavigation <> iConfigVisuNavigation) OR (rEnableConfigMaxToolLength <> rConfigMaxToolLength)  THEN
			xChkConfigStation:=TRUE;
			ptrTFunction^.xStop:=NOT(ptrTFunction^.xEnd);
			IF ptrTFunction^.xEnd THEN
				ptrTFunction^.xStart:=FALSE;
			END_IF;
		END_IF;
	END_IF;
	IF xChkConfigStation THEN
		IF ptrTFunction^.xEnd THEN
			IF (iEnableConfigMachineType <> iConfigMachineType) THEN
				ptrTFunction^.iErrorNr:=7001;	(* Error-->Config Machine Type changed *)
			END_IF;
			IF (iEnableConfigAxisType <> iConfigAxisType) THEN
				ptrTFunction^.iErrorNr:=7002;	(* Error-->Config Axis Type changed *)
			END_IF;
			IF (iEnableConfigVisuNavigation <> iConfigVisuNavigation) THEN
				TStation.TControl.diErrorNr:=7003;	(* Error-->Config Visu Navigation changed *)
			END_IF;
			IF (rEnableConfigMaxToolLength <> rConfigMaxToolLength) THEN
				TStation.TControl.diErrorNr:=7004;	(* Error-->Config Max Tool Length changed *)
			END_IF;
			xStartFunction:=FALSE;
			xChkConfigStation:=FALSE;
			xStationError:=TRUE;
			RETURN;
		END_IF;
	END_IF;
END_IF;
(******************************************************************************************************************************************)
(****************************				              Funktionen                                                               *****************************)
(******************************************************************************************************************************************)
IF xStartFunction AND NOT(xSetEnd) THEN
	IF (iStationFunctionNr = 1) THEN
		FBFctToolFeedReference(	xMicroRodActive:= xMicroRodActive,
								xBeckhoffDriveActive:= xBeckhoffDriveActive,
								xSafetyCircuitOn:= xSafetyCircuitOn1 AND xSafetyCircuitOn2,
								T_Standard:= T_Standard,
								xStart:= ptrTFunction^.xStart,
								xReset:=ptrTFunction^.xReset,
								xStop:= ptrTFunction^.xStop,
								xQuitErr:= ptrTFunction^.xQuitErr,
								xAbord:= ptrTFunction^.xAbord,
								TAxisToolFeeder:= ptrTAxisToolFeeder^,
								xEnd=>ptrTFunction^.xEnd,
								xError=>ptrTFunction^.xError,
								iErrorNr=>ptrTFunction^.iErrorNr);
	END_IF;
	IF (iStationFunctionNr = 2) THEN
		FBFctToolRotationTorqueStart(	xMicroRodActive:= xMicroRodActive,
									xBeckhoffDriveActive:= xBeckhoffDriveActive,
									xSafetyCircuitOn:=xSafetyCircuitOn1 AND xSafetyCircuitOn2,
									xStart:= ptrTFunction^.xStart,
									xReset:=ptrTFunction^.xReset,
									xStop:= ptrTFunction^.xStop,
									xQuitErr:= ptrTFunction^.xQuitErr,
									xAbord:= ptrTFunction^.xAbord,
									TAxisToolLeft:= ptrTAxisToolLeft^,
									TAxisToolCenter:= ptrTAxisToolCenter^,
									TAxisToolRight:=ptrTAxisToolRight^,
									TAxisToolFeeder:=ptrTAxisToolFeeder^,
									xEnd=>ptrTFunction^.xEnd,
									xError=>ptrTFunction^.xError,
									iErrorNr=>ptrTFunction^.iErrorNr);
	END_IF;
	IF (iStationFunctionNr = 3) THEN
		FBFctToolRotationTorqueStop(	xMicroRodActive:= xMicroRodActive,
									xBeckhoffDriveActive:= xBeckhoffDriveActive,
									xSafetyCircuitOn:=xSafetyCircuitOn1 AND xSafetyCircuitOn2,
									xStart:= ptrTFunction^.xStart,
									xReset:=ptrTFunction^.xReset,
									xStop:= ptrTFunction^.xStop,
									xQuitErr:= ptrTFunction^.xQuitErr,
									xAbord:= ptrTFunction^.xAbord,
									TAxisToolLeft:= ptrTAxisToolLeft^,
									TAxisToolCenter:= ptrTAxisToolCenter^,
									TAxisToolRight:=ptrTAxisToolRight^,
									TAxisToolFeeder:=ptrTAxisToolFeeder^,
									xEnd=>ptrTFunction^.xEnd,
									xError=>ptrTFunction^.xError,
									iErrorNr=>ptrTFunction^.iErrorNr);
	END_IF;
	IF (iStationFunctionNr = 4) OR (iStationFunctionNr = 5) THEN
		FBFctGrindFeedAbsRelPosition(	xMicroRodActive:= xMicroRodActive,
										xBeckhoffDriveActive:= xBeckhoffDriveActive,
										xSafetyCircuitOn:= xSafetyCircuitOn1 AND xSafetyCircuitOn2,
										iFunctionNr:= iStationFunctionNr,
										xStart:= ptrTFunction^.xStart,
										xReset:=ptrTFunction^.xReset,
										xStop:= ptrTFunction^.xStop,
										xQuitErr:= ptrTFunction^.xQuitErr,
										xAbord:= ptrTFunction^.xAbord,
										TAxisGrindFeeder:= ptrTAxisGrindFeeder^,
										xEnd=>ptrTFunction^.xEnd,
										xError=>ptrTFunction^.xError,
										iErrorNr=>ptrTFunction^.iErrorNr);
	END_IF;
	IF (iStationFunctionNr >= 6) AND (iStationFunctionNr <= 10) THEN
		FBFctSetAxisPosition(	xMicroRodActive:= xMicroRodActive,
							xBeckhoffDriveActive:= xBeckhoffDriveActive,
							xSafetyCircuitOn:= xSafetyCircuitOn1 AND xSafetyCircuitOn2,
							iFunctionNr:= iStationFunctionNr,
							xStart:= ptrTFunction^.xStart,
							xReset:=ptrTFunction^.xReset,
							xStop:= ptrTFunction^.xStop,
							xQuitErr:= ptrTFunction^.xQuitErr,
							xAbord:= ptrTFunction^.xAbord,
							TAxisToolLeft:= ptrTAxisToolLeft^,
							TAxisToolCenter:= ptrTAxisToolCenter^,
							TAxisToolRight:=ptrTAxisToolRight^,
							TAxisToolFeeder:=ptrTAxisToolFeeder^,
							TAxisGrindFeeder:= ptrTAxisGrindFeeder^,
							xEnd=>ptrTFunction^.xEnd,
							xError=>ptrTFunction^.xError,
							iErrorNr=>ptrTFunction^.iErrorNr);
	END_IF;
	IF (iStationFunctionNr = 11) THEN
		(* AutoGeometry *)
		FBFctToolWorkingGeometry(	xMicroRodActive:= xMicroRodActive,
									xBeckhoffDriveActive:= xBeckhoffDriveActive,
									xSafetyCircuitOn:= xSafetyCircuitOn1 AND xSafetyCircuitOn2,
									T_ProcessImageData:= T_ProcessImageData,
									T_Standard:= T_Standard,
									xStart:= ptrTFunction^.xStart,
									xReset:=ptrTFunction^.xReset,
									xStop:= ptrTFunction^.xStop,
									xQuitErr:= ptrTFunction^.xQuitErr,
									xAbord:= ptrTFunction^.xAbord,
									TAxisToolLeft:= ptrTAxisToolLeft^,
									TAxisToolCenter:= ptrTAxisToolCenter^,
									TAxisToolRight:=ptrTAxisToolRight^,
									TAxisToolFeeder:=ptrTAxisToolFeeder^,
									TAxisGrindFeeder:= ptrTAxisGrindFeeder^,
									T_WorkTool:=TStation.T_WorkTool,
									xEnd=>ptrTFunction^.xEnd,
									xError=>ptrTFunction^.xError,
									iErrorNr=>ptrTFunction^.iErrorNr,
									bActivePartNumber=>bActivePartNumber,
									lrProcessToolFeederActualPosition=>lrProcessToolFeederActualPosition,
									lrProcessToolFeederSpeed=>lrProcessToolFeederSpeed,
									iCountDownPlungeCycle=>TStation.TControl.iCountDownPlungeCycle);
	END_IF;
	IF (iStationFunctionNr = 12) THEN
		(* AutoGroove *)
		FBFctToolWorkingGroove(		xMicroRodActive:= xMicroRodActive,
									xBeckhoffDriveActive:= xBeckhoffDriveActive,
									xSafetyCircuitOn:= xSafetyCircuitOn1 AND xSafetyCircuitOn2,
									xDoNotMoveGrindPosition:=T_ProcessImageData.T_AutoGroovePara.xBlockGrindFeeder,
									T_ProcessImageData:= T_ProcessImageData,
									T_Standard:= T_Standard,
									xStart:= ptrTFunction^.xStart,
									xReset:=ptrTFunction^.xReset,
									xStop:= ptrTFunction^.xStop,
									xQuitErr:= ptrTFunction^.xQuitErr,
									xAbord:= ptrTFunction^.xAbord,
									TAxisToolLeft:= ptrTAxisToolLeft^,
									TAxisToolCenter:= ptrTAxisToolCenter^,
									TAxisToolRight:=ptrTAxisToolRight^,
									TAxisToolFeeder:=ptrTAxisToolFeeder^,
									TAxisGrindFeeder:= ptrTAxisGrindFeeder^,
									T_WorkTool:=TStation.T_WorkTool,
									rStartPosAutoGrooveToolRotation:=TStation.rStartPosAutoGrooveToolRotation,
									xEnd=>ptrTFunction^.xEnd,
									xError=>ptrTFunction^.xError,
									iErrorNr=>ptrTFunction^.iErrorNr,
									bActivePartNumber=>bActivePartNumber,
									lrProcessToolFeederActualPosition=>lrProcessToolFeederActualPosition,
									lrProcessToolFeederSpeed=>lrProcessToolFeederSpeed);
	END_IF;
	IF (iStationFunctionNr = 13) THEN
		FBFctToolCalibration(			xMicroRodActive:= xMicroRodActive,
									xBeckhoffDriveActive:= xBeckhoffDriveActive,
									xSafetyCircuitOn:= xSafetyCircuitOn1 AND xSafetyCircuitOn2,
									T_ProcessImageData:= T_ProcessImageData,
									T_Standard:= T_Standard,
									xStart:= ptrTFunction^.xStart,
									xReset:=ptrTFunction^.xReset,
									xStop:= ptrTFunction^.xStop,
									xQuitErr:= ptrTFunction^.xQuitErr,
									xAbord:= ptrTFunction^.xAbord,
									TAxisToolLeft:= ptrTAxisToolLeft^,
									TAxisToolCenter:= ptrTAxisToolCenter^,
									TAxisToolRight:=ptrTAxisToolRight^,
									TAxisToolFeeder:=ptrTAxisToolFeeder^,
									TAxisGrindFeeder:= ptrTAxisGrindFeeder^,
									T_WorkTool:=TStation.T_WorkTool,
									xEnd=>ptrTFunction^.xEnd,
									xError=>ptrTFunction^.xError,
									iErrorNr=>ptrTFunction^.iErrorNr,
									lrProcessToolFeederActualPosition=>lrProcessToolFeederActualPosition,
									lrProcessToolFeederSpeed=>lrProcessToolFeederSpeed);
	END_IF;
	IF (iStationFunctionNr = 14) OR (iStationFunctionNr = 15) THEN
		FBFctToolFeedAbsRelPosition(		xMicroRodActive:= xMicroRodActive,
										xBeckhoffDriveActive:= xBeckhoffDriveActive,
										xSafetyCircuitOn:= xSafetyCircuitOn1 AND xSafetyCircuitOn2,
										iFunctionNr:= iStationFunctionNr,
										xStart:= ptrTFunction^.xStart,
										xReset:=ptrTFunction^.xReset,
										xStop:= ptrTFunction^.xStop,
										xQuitErr:= ptrTFunction^.xQuitErr,
										xAbord:= ptrTFunction^.xAbord,
										TAxisToolFeeder:= ptrTAxisToolFeeder^,
										xEnd=>ptrTFunction^.xEnd,
										xError=>ptrTFunction^.xError,
										iErrorNr=>ptrTFunction^.iErrorNr);
	END_IF;
	IF (iStationFunctionNr = 16) OR (iStationFunctionNr = 17) THEN
		FBFctSwitchOnOffPowerSupply(	xMicroRodActive:= xMicroRodActive,
									xBeckhoffDriveActive:= xBeckhoffDriveActive,
									xSafetyCircuitOn:= xSafetyCircuitOn1 AND xSafetyCircuitOn2,
									iFunctionNr:= iStationFunctionNr,
									xStart:= ptrTFunction^.xStart,
									xReset:=ptrTFunction^.xReset,
									xStop:= ptrTFunction^.xStop,
									xQuitErr:= ptrTFunction^.xQuitErr,
									xAbord:= ptrTFunction^.xAbord,
									TAxisToolLeft:= ptrTAxisToolLeft^,
									TAxisToolCenter:= ptrTAxisToolCenter^,
									TAxisToolRight:=ptrTAxisToolRight^,
									TAxisToolFeeder:=ptrTAxisToolFeeder^,
									TAxisGrindFeeder:= ptrTAxisGrindFeeder^,
									TAxisGrindSpindle:= ptrTAxisGrindSpindle^,
									xEnd=>ptrTFunction^.xEnd,
									xError=>ptrTFunction^.xError,
									iErrorNr=>ptrTFunction^.iErrorNr);
	END_IF;
	IF (iStationFunctionNr = 18) THEN
		FBFctStopAxisMovement(	xMicroRodActive:= xMicroRodActive,
								xBeckhoffDriveActive:= xBeckhoffDriveActive,
								xSafetyCircuitOn:= xSafetyCircuitOn1 AND xSafetyCircuitOn2,
								T_ProcessImageData:= T_ProcessImageData,
								T_Standard:= T_Standard,
								xStart:= ptrTFunction^.xStart,
								xReset:=ptrTFunction^.xReset,
								xStop:= ptrTFunction^.xStop,
								xQuitErr:= ptrTFunction^.xQuitErr,
								xAbord:= ptrTFunction^.xAbord,
								TAxisToolLeft:= ptrTAxisToolLeft^,
								TAxisToolCenter:= ptrTAxisToolCenter^,
								TAxisToolRight:=ptrTAxisToolRight^,
								TAxisToolFeeder:=ptrTAxisToolFeeder^,
								TAxisGrindFeeder:= ptrTAxisGrindFeeder^,
								TAxisGrindSpindle:= ptrTAxisGrindSpindle^,
								xEnd=>ptrTFunction^.xEnd,
								xError=>ptrTFunction^.xError,
								iErrorNr=>ptrTFunction^.iErrorNr);
	END_IF;
	IF (iStationFunctionNr = 19) THEN
		(* AutoGeometryMultiCycle*)
		FBFctToolWorkingGeometryMultiCycle(	xMicroRodActive:= xMicroRodActive,
											xBeckhoffDriveActive:= xBeckhoffDriveActive,
											xSafetyCircuitOn:= xSafetyCircuitOn1 AND xSafetyCircuitOn2,
											T_ProcessImageData:= T_ProcessImageData,
											T_Standard:= T_Standard,
											xStart:= ptrTFunction^.xStart,
											xReset:=ptrTFunction^.xReset,
											xStop:= ptrTFunction^.xStop,
											xQuitErr:= ptrTFunction^.xQuitErr,
											xAbord:= ptrTFunction^.xAbord,
											TAxisToolLeft:= ptrTAxisToolLeft^,
											TAxisToolCenter:= ptrTAxisToolCenter^,
											TAxisToolRight:=ptrTAxisToolRight^,
											TAxisToolFeeder:=ptrTAxisToolFeeder^,
											TAxisGrindFeeder:= ptrTAxisGrindFeeder^,
											T_WorkTool:=TStation.T_WorkTool,
											xEnd=>ptrTFunction^.xEnd,
											xError=>ptrTFunction^.xError,
											iErrorNr=>ptrTFunction^.iErrorNr,
											bActivePartNumber=>bActivePartNumber,
											lrProcessToolFeederActualPosition=>lrProcessToolFeederActualPosition,
											lrProcessToolFeederSpeed=>lrProcessToolFeederSpeed,
											iCountDownPlungeCycle=>TStation.TControl.iCountDownPlungeCycle);
	END_IF;
	(* 17.11.2010: KFS 	{	*)
	IF (iStationFunctionNr = 20) THEN
		FBFctToolFeedMaxLenReference(	xMicroRodActive:= xMicroRodActive,
										xBeckhoffDriveActive:= xBeckhoffDriveActive,
										xSafetyCircuitOn:= xSafetyCircuitOn1 AND xSafetyCircuitOn2,
										T_Standard:= T_Standard,
										xStart:= ptrTFunction^.xStart,
										xReset:=ptrTFunction^.xReset,
										xStop:= ptrTFunction^.xStop,
										xQuitErr:= ptrTFunction^.xQuitErr,
										xAbord:= ptrTFunction^.xAbord,
										TAxisToolFeeder:= ptrTAxisToolFeeder^,
										xEnd=>ptrTFunction^.xEnd,
										xError=>ptrTFunction^.xError,
										iErrorNr=>ptrTFunction^.iErrorNr);
	END_IF;
	(* 17.11.2010: KFS 	{	*)
END_IF;
(******************************************************************************************************************************************)
(****************************				         Init / Reset Hardware                                                 *****************************)
(******************************************************************************************************************************************)
IF xSetEnd THEN
	xStationError:=FALSE;
	xInitError:=FALSE;
	xInitStart:=FALSE;
	xInitStop:=FALSE;
	xInitStep:=FALSE;
	xSetEnd:=FALSE;
	xTmpStart:=FALSE;
	TStation.TControl.xEnd:=TRUE;
	TStation.TControl.xStart:=FALSE;
	TStation.TControl.xStop:=FALSE;
	TStation.TControl.xAbord:=FALSE;
	IF NOT(xDontDeleteErrorFlag) THEN
		TStation.TControl.xError:=FALSE;
		TStation.TControl.diErrorNr:=0;
	END_IF;
	xDontDeleteErrorFlag:=FALSE;
	xStartFunction:=FALSE;
	iStepError:=100;
	xStepError:=FALSE;
	xTmpStationError:=FALSE;
	xChkConfigStation:=FALSE;
	diErrorNumber:=0;
	xSetError:=FALSE;
	xReadyToQuitErr:=FALSE;
END_IF;
(*03.03.2017: KFS { *)
IF T_StartUp.T_State.xCompleted THEN
	IF ptrTCylToolLeftActive^.T_CtrleCyl.T_Standard.xActivOn AND ptrTAxisToolLeft^.T_CtrleSingle.xPower
	     AND NOT(ptrTAxisToolLeft^.T_CtrleSingle.xExecute) AND ptrTAxisToolLeft^.T_CtrleSingle.xDone THEN
		ptrTAxisToolLeft^.T_CtrleSingle.iFunction:=4;
		ptrTAxisToolLeft^.T_CtrleSingle.xExecute:=TRUE;
	END_IF;
	IF ptrTCylToolRightActive^.T_CtrleCyl.T_Standard.xActivOn AND ptrTAxisToolRight^.T_CtrleSingle.xPower
	     AND NOT(ptrTAxisToolRight^.T_CtrleSingle.xExecute) AND ptrTAxisToolRight^.T_CtrleSingle.xDone THEN
		ptrTAxisToolRight^.T_CtrleSingle.iFunction:=4;
		ptrTAxisToolRight^.T_CtrleSingle.xExecute:=TRUE;
	END_IF;
END_IF;
(*03.03.2017: KFS } *)
END_FUNCTION_BLOCK
ACTION CtrlDisableStation:
(******************************************************************************************************************************************)
(****************************				                Disable Part                                                            *****************************)
(******************************************************************************************************************************************)
fbFTrig(CLK:=TStation.TControl.xEnable);
IF fbFTrig.Q THEN
	xInitSetEnable:=FALSE;
	xInitDelEnable:=FALSE;
	xRdyDisableStation:=FALSE;
END_IF;
IF (fbFTrig.Q OR xInitDelEnable) THEN
	IF NOT(xInitDelEnable) OR fbFTrig.Q THEN
		xReadyChkError:=FALSE;
		TStation.TControl.xEnd:=FALSE;
		IF NOT(xDontDeleteErrorFlag) THEN
			TStation.TControl.xError:=FALSE;
		END_IF;
		xInitDelEnable:=TRUE;
		TStation.TControl.xRdy:=FALSE;
		iStepEnable:=100;
		iAxisFunctionNr:=1;
		iStationFunctionNr:=1;
		xInitStep:=FALSE;
	END_IF;
	CASE iStepEnable OF
		100:	IF NOT(xInitStep) THEN
				xInitStep:=TRUE;
				xSetEnableConfig:=FALSE;
				xStartFunction:=TRUE;
				ptrTFunction^.xReset:=TRUE;
			END_IF;
			IF NOT(ptrTFunction^.xReset) AND ptrTFunction^.xEnd THEN
				(* Alle Funktionen Resetten *)
				IF (iStationFunctionNr < iMaxFunctionNr) THEN
					iStationFunctionNr:=iStationFunctionNr + 1;
					ptrTFunction^.xReset:=TRUE;
				ELSE
					xInitStep:=FALSE;
					xStartFunction:=FALSE;
					iStepEnable:=200;
				END_IF;
			END_IF;
		200:	IF NOT(xInitStep) THEN
				xInitStep:=TRUE;
				IF TStation.TControl.xHardwareConfigError THEN
					TStation.TControl.xHardwareConfigError:=FALSE;
					TStation.TControl.xActiveHardware:=FALSE;
				ELSE
					xInitStep:=FALSE;
					iStepEnable:=300;
				END_IF;
				RETURN;
			END_IF;
			IF NOT(TStation.TControl.xError) OR xDontDeleteErrorFlag THEN
				TStation.TControl.xActiveHardware:=TRUE;
				xInitStep:=FALSE;
				iStepEnable:=300;
				RETURN;
			END_IF;
		300:	IF NOT(xInitStep) THEN	(* Alle Hardware Bausteine resetten *)
				xInitStep:=TRUE;
				ptrTCylToolTension^.T_CtrleCyl.xFBActiv:=FALSE;
				(*22.12.2009: KFS {    *)
				IF xMicroRodActive THEN
					ptrTCylToolLeftActive^.T_CtrleCyl.xFBActiv:=FALSE;
					ptrTCylToolRightActive^.T_CtrleCyl.xFBActiv:=FALSE;
					ptrTCylToolCenterActive^.T_CtrleCyl.xFBActiv:=FALSE;
					ptrTCylToolPrismaLeftActive^.T_CtrleCyl.xFBActiv:=FALSE;
					ptrTCylToolPrismaRightActive^.T_CtrleCyl.xFBActiv:=FALSE;
					ptrTToolFeederWorkLength^.T_CtrleCyl.xFBActiv:=FALSE;
				END_IF;
				(*22.12.2009: KFS }   *)
				IF xBeckhoffDriveActive THEN
					ptrTAxisToolLeft^.T_CtrleSingle.xReset:=TRUE;
					IF xMicroRodActive THEN
						ptrTAxisToolCenter^.T_CtrleSingle.xReset:=TRUE;
					END_IF;
					ptrTAxisToolRight^.T_CtrleSingle.xReset:=TRUE;
					ptrTAxisToolFeeder^.T_CtrleSingle.xReset:=TRUE;
					ptrTAxisGrindFeeder^.T_CtrleSingle.xReset:=TRUE;
					ptrTAxisGrindSpindle^.T_CtrleSingle.xReset:=TRUE;
				ELSE
					TStation.TControl.xResetHardware:=TRUE;
					iStepEnable:=399;
					RETURN;
				END_IF;
			END_IF;
			IF xTmp THEN
				RETURN;	(* Wait until all Drives finished *)
			END_IF;
			IF (NOT(ptrTAxisToolLeft^.T_CtrleSingle.xReset) AND ptrTAxisToolLeft^.T_CtrleSingle.xErr) OR
			    (((NOT(ptrTAxisToolCenter^.T_CtrleSingle.xReset) AND ptrTAxisToolCenter^.T_CtrleSingle.xErr AND xMicroRodActive) OR NOT(xMicroRodActive))) OR
			    (NOT(ptrTAxisToolRight^.T_CtrleSingle.xReset) AND ptrTAxisToolRight^.T_CtrleSingle.xErr) OR
			    (NOT(ptrTAxisToolFeeder^.T_CtrleSingle.xReset) AND ptrTAxisToolFeeder^.T_CtrleSingle.xErr)OR
			    (NOT(ptrTAxisGrindFeeder^.T_CtrleSingle.xReset) AND ptrTAxisGrindFeeder^.T_CtrleSingle.xErr) OR
			    (NOT(ptrTAxisGrindSpindle^.T_CtrleSingle.xReset) AND ptrTAxisGrindSpindle^.T_CtrleSingle.xErr) THEN
				xInitStep:=FALSE;
				iStepEnable:=400;
			END_IF;
			IF NOT(ptrTAxisToolLeft^.T_CtrleSingle.xReset) AND ptrTAxisToolLeft^.T_CtrleSingle.xDone AND
			    ((NOT(ptrTAxisToolCenter^.T_CtrleSingle.xReset) AND ptrTAxisToolCenter^.T_CtrleSingle.xDone AND xMicroRodActive) OR NOT(xMicroRodActive)) AND
			    NOT(ptrTAxisToolRight^.T_CtrleSingle.xReset) AND ptrTAxisToolRight^.T_CtrleSingle.xDone AND
			    NOT(ptrTAxisToolFeeder^.T_CtrleSingle.xReset) AND ptrTAxisToolFeeder^.T_CtrleSingle.xDone AND
			    NOT(ptrTAxisGrindFeeder^.T_CtrleSingle.xReset) AND ptrTAxisGrindFeeder^.T_CtrleSingle.xDone AND
			    NOT(ptrTAxisGrindSpindle^.T_CtrleSingle.xReset) AND ptrTAxisGrindSpindle^.T_CtrleSingle.xDone THEN
				TStation.TControl.xActiveHardware:=FALSE;
				xInitStep:=FALSE;
				xInitDelEnable:=FALSE;
				xSetEnd:=TRUE;
				xRdyDisableStation:=TRUE;
			END_IF;
		399:	IF NOT(TStation.TControl.xResetHardware) THEN
				TStation.TControl.xActiveHardware:=FALSE;
				xInitStep:=FALSE;
				xInitDelEnable:=FALSE;
				xSetEnd:=TRUE;
				xRdyDisableStation:=TRUE;
			END_IF;
		400:	IF NOT(xInitStep) THEN
				xInitStep:=TRUE;
				ptrTAxisToolLeft^.T_CtrleSingle.iFunction:=1;
				ptrTAxisToolLeft^.T_CtrleSingle.xExecute:=ptrTAxisToolLeft^.T_CtrleSingle.xErr;
				IF xMicroRodActive THEN
					ptrTAxisToolCenter^.T_CtrleSingle.iFunction:=1;
					ptrTAxisToolCenter^.T_CtrleSingle.xExecute:=ptrTAxisToolCenter^.T_CtrleSingle.xErr;
				END_IF;
				ptrTAxisToolRight^.T_CtrleSingle.iFunction:=1;
				ptrTAxisToolRight^.T_CtrleSingle.xExecute:=ptrTAxisToolRight^.T_CtrleSingle.xErr;
				ptrTAxisToolFeeder^.T_CtrleSingle.iFunction:=1;
				ptrTAxisToolFeeder^.T_CtrleSingle.xExecute:=ptrTAxisToolFeeder^.T_CtrleSingle.xErr;
				ptrTAxisGrindFeeder^.T_CtrleSingle.iFunction:=1;
				ptrTAxisGrindFeeder^.T_CtrleSingle.xExecute:=ptrTAxisGrindFeeder^.T_CtrleSingle.xErr;
				ptrTAxisGrindSpindle^.T_CtrleSingle.iFunction:=1;
				ptrTAxisGrindSpindle^.T_CtrleSingle.xExecute:=ptrTAxisGrindSpindle^.T_CtrleSingle.xErr;
			END_IF;
			IF xTmp THEN
				RETURN;	(* Wait until all Drives finished *)
			END_IF;
			IF NOT(ptrTAxisToolLeft^.T_CtrleSingle.xExecute) AND ptrTAxisToolLeft^.T_CtrleSingle.xErr AND
			    ((NOT(ptrTAxisToolCenter^.T_CtrleSingle.xExecute) AND ptrTAxisToolCenter^.T_CtrleSingle.xErr AND xMicroRodActive) OR NOT(xMicroRodActive)) AND
			    NOT(ptrTAxisToolRight^.T_CtrleSingle.xExecute) AND ptrTAxisToolRight^.T_CtrleSingle.xErr AND
			    NOT(ptrTAxisToolFeeder^.T_CtrleSingle.xExecute) AND ptrTAxisToolFeeder^.T_CtrleSingle.xErr AND
			    NOT(ptrTAxisGrindFeeder^.T_CtrleSingle.xExecute) AND ptrTAxisGrindFeeder^.T_CtrleSingle.xErr AND
			    NOT(ptrTAxisGrindSpindle^.T_CtrleSingle.xExecute) AND ptrTAxisGrindSpindle^.T_CtrleSingle.xErr THEN
				xInitStep:=FALSE;
				iStepEnable:=500;
			END_IF;
			IF NOT(ptrTAxisToolLeft^.T_CtrleSingle.xExecute) AND ptrTAxisToolLeft^.T_CtrleSingle.xDone AND
			    ((NOT(ptrTAxisToolCenter^.T_CtrleSingle.xExecute) AND ptrTAxisToolCenter^.T_CtrleSingle.xDone AND xMicroRodActive) OR NOT(xMicroRodActive)) AND
			    NOT(ptrTAxisToolRight^.T_CtrleSingle.xExecute) AND ptrTAxisToolRight^.T_CtrleSingle.xDone AND
			    NOT(ptrTAxisToolFeeder^.T_CtrleSingle.xExecute) AND ptrTAxisToolFeeder^.T_CtrleSingle.xDone AND
			    NOT(ptrTAxisGrindFeeder^.T_CtrleSingle.xExecute) AND ptrTAxisGrindFeeder^.T_CtrleSingle.xDone AND
			    NOT(ptrTAxisGrindSpindle^.T_CtrleSingle.xExecute) AND ptrTAxisGrindSpindle^.T_CtrleSingle.xDone THEN
				TStation.TControl.xActiveHardware:=FALSE;
				xInitStep:=FALSE;
				xInitDelEnable:=FALSE;
				xSetEnd:=TRUE;
				xRdyDisableStation:=TRUE;
			END_IF;
		500:	TStation.TControl.xActiveHardware:=FALSE;
			TStation.TControl.diErrorNr:=8000000 + 10;	(* Station Disable Fehlerhaft *)
			TStation.TControl.xError:=TRUE;
			xDontDeleteErrorFlag:=TRUE;
			xInitStep:=FALSE;
			xInitDelEnable:=FALSE;
			xSetEnd:=TRUE;
			xRdyDisableStation:=TRUE;
	END_CASE;
END_IF;
END_ACTION
ACTION CtrlEnableStation:
(******************************************************************************************************************************************)
(****************************				                Enable Part                                                            *****************************)
(******************************************************************************************************************************************)
fbRTrig(CLK:=TStation.TControl.xEnable);
IF fbRTrig.Q THEN
	xInitSetEnable:=FALSE;
	xInitDelEnable:=FALSE;
END_IF;
IF (fbRTrig.Q OR xInitSetEnable) THEN
	IF NOT(fbRTrig.Q) AND xReadyChkError THEN
		IF xSetError OR ptrTAxisToolLeft^.T_CtrleSingle.xErr OR (ptrTAxisToolCenter^.T_CtrleSingle.xErr AND xMicroRodActive) OR
		     ptrTAxisToolRight^.T_CtrleSingle.xErr OR ptrTAxisToolFeeder^.T_CtrleSingle.xErr OR ptrTAxisGrindFeeder^.T_CtrleSingle.xErr THEN
			IF (xTmp OR (NOT(T_BoxID.T_Ctrle.xErr) AND NOT(T_BoxID.T_Ctrle.xDone))) AND NOT(xSetError) THEN
				RETURN;	(* Wait until all Actuators are not working *)
			END_IF;
			IF xSetError THEN
				xSetError:=FALSE;
				TStation.TControl.diErrorNr:=8000000 + diErrorNumber;
			ELSE
				ptrTAxisToolLeft^.T_CtrleSingle.xReset:=ptrTAxisToolLeft^.T_CtrleSingle.xErr;
				IF xMicroRodActive THEN
					ptrTAxisToolCenter^.T_CtrleSingle.xReset:=ptrTAxisToolCenter^.T_CtrleSingle.xErr;
				END_IF;
				ptrTAxisToolRight^.T_CtrleSingle.xReset:=ptrTAxisToolRight^.T_CtrleSingle.xErr;
				ptrTAxisToolFeeder^.T_CtrleSingle.xReset:=ptrTAxisToolFeeder^.T_CtrleSingle.xErr;
				ptrTAxisGrindFeeder^.T_CtrleSingle.xReset:=ptrTAxisGrindFeeder^.T_CtrleSingle.xErr;
				T_BoxID.T_Ctrle.xReset:=T_BoxID.T_Ctrle.xErr;
				IF ptrTAxisToolLeft^.T_CtrleSingle.xErr THEN TStation.TControl.diErrorNr:=1000000 + ptrTAxisToolLeft^.T_CtrleSingle.udiErrorID; END_IF;
				IF xMicroRodActive THEN
					IF ptrTAxisToolCenter^.T_CtrleSingle.xErr THEN TStation.TControl.diErrorNr:=2000000 + ptrTAxisToolCenter^.T_CtrleSingle.udiErrorID; END_IF;
				END_IF;
				IF ptrTAxisToolRight^.T_CtrleSingle.xErr THEN TStation.TControl.diErrorNr:=3000000 + ptrTAxisToolRight^.T_CtrleSingle.udiErrorID; END_IF;
				IF ptrTAxisToolFeeder^.T_CtrleSingle.xErr THEN TStation.TControl.diErrorNr:=4000000 + ptrTAxisToolFeeder^.T_CtrleSingle.udiErrorID; END_IF;
				IF ptrTAxisGrindFeeder^.T_CtrleSingle.xErr THEN TStation.TControl.diErrorNr:=5000000 + ptrTAxisGrindFeeder^.T_CtrleSingle.udiErrorID; END_IF;
				IF T_BoxID.T_Ctrle.xErr THEN TStation.TControl.diErrorNr:=7000000 + T_BoxID.T_Ctrle.udiErrorID; END_IF;
			END_IF;
			TStation.TControl.xEnable:=FALSE;
			TStation.TControl.xError:=TRUE;
			xDontDeleteErrorFlag:=TRUE;
			RETURN;
		END_IF;
	END_IF;
	IF NOT(xInitSetEnable) OR fbRTrig.Q THEN
		xSetEnd:=FALSE;
		xInitSetEnable:=TRUE;
		TStation.TControl.xRdy:=FALSE;
		TStation.TControl.xEnd:=FALSE;
		TStation.TControl.xError:=FALSE;
		TStation.TControl.diErrorNr:=0;
		iStepEnable:=100;
		iAxisFunctionNr:=1;
		iStationFunctionNr:=1;
		xSetEnableConfig:=FALSE;
		xInitStep:=FALSE;
		RETURN;
	END_IF;
	CASE iStepEnable OF
		100:	IF NOT(xRdyDisableStation) THEN
				iStepEnable:=110;
				RETURN;
			END_IF;
			IF NOT(xInitStep) THEN
				xInitStep:=TRUE;
				xStartFunction:=TRUE;
				ptrTFunction^.xReset:=TRUE;
				(* Initialisierung der HW *)
				TStation.TControl.xActiveHardware:=TRUE;
				TStation.T_MachineConfig.iConfigMachineType:=iConfigMachineType;
				TStation.T_MachineConfig.iConfigAxisType:=iConfigAxisType;
				TStation.T_MachineConfig.iConfigVisuNavigation:=iConfigVisuNavigation;
				TStation.T_MachineConfig.rConfigMaxToolLength:=rConfigMaxToolLength;
				(* Initialisierung der Aktuatoren *)

